{attribute 'linkalways'} 
{attribute 'no_explicit_call' := 'This FB is a CLASS and must be accessed using methods or properties'}
{attribute 'enable_dynamic_creation'}
{attribute 'TcRpcEnable'}
FUNCTION_BLOCK RpcServer EXTENDS Server
VAR
	rpcServerConfig : RpcServerConfigV1;
	rpcHandlers : RpcHandlers;
	rpcManager : RpcManager(rpcHandlers, rpcServerConfig);
	rpcMiddleware : RpcMiddleware(rpcManager);
END_VAR

METHOD FB_init : BOOL
VAR_INPUT
	bInitRetains : BOOL; // if TRUE, the retain variables are initialized (warm start / cold start)
	bInCopyCode : BOOL;  // if TRUE, the instance afterwards gets moved into the copy code (online change)
END_VAR
MiddlewareStack.Use(rpcMiddleware);
END_METHOD

PROPERTY PUBLIC Rpc : I_RpcHandlers
GET
Rpc := rpcHandlers;
END_GET
END_PROPERTY

END_FUNCTION_BLOCK

(* stored: Version 1.1.0.1, ProductVersion 3.1.4024.12
   POU RpcServer: Id {a6ca3c86-e0c6-4dcd-95d3-86401e8307e7}, SpecialFunc None
   Folder Constructor: Id {63db7c18-245f-4309-a927-a9a0d3af3475}
   Method FB_init: Id {d6649ca6-46cd-40bd-9987-0427348a48b4}
   Property Rpc: Id {a0185c7a-0cf4-4ff1-928a-6e9738b941cb}
   Get Get: Id {5740807a-491f-42b5-b2df-f076c59269a5} *)
